FUNCTION FILETIME_TO_TOD : TIME_OF_DAY //Converts 64bit T_FILETIME to TIME_OF_DAY (TOD#15:36:30.123)
VAR_INPUT
	IN														: T_FILETIME;
END_VAR
VAR
END_VAR

FILETIME_TO_TOD												:= SYSTEMTIME_TO_TOD(FILETIME_TO_SYSTEMTIME(IN));

END_FUNCTION

(* stored: Version 1.1.0.1, ProductVersion 3.1.4024.3
   POU FILETIME_TO_TOD: Id {2dfd0802-d1df-4ed2-8352-86631f3e5384}, SpecialFunc None *)
